(* IEC 61131-3 sources: POMIRTS_lab3/AS/Library_2/MTLoadSim/V1.01.0, 3 files *)

(* ---- MTLoadSim.typ ---- *)
(********************************************************************
 * COPYRIGHT -- Bernecker + Rainer
 ********************************************************************
 * Library: MTLoadSim
 * File: MTLoadSim.typ
 * Author: B + R
 ********************************************************************
 * Data types of library MTLoadSim
 ********************************************************************)

TYPE
	MTLoadSimConfigFrictionType : 	STRUCT
		Mode : MTLoadSimFricModeEnum;
		StaticFriction : REAL;
		DynamicFriction : REAL;
		ViscousFriction : REAL;
		StribeckVelocity : REAL;
		ApproximateVelocity : REAL;
		FrictionEpsilon : REAL;
		StribeckExponent : REAL;
	END_STRUCT;
	MTLoadSimConfigMassType : 	STRUCT
		Inertia : REAL;
		InitialStates : ARRAY[0..1]OF REAL;
	END_STRUCT;
	MTLoadSimConfigTwoMassType : 	STRUCT
		InertiaMass1 : REAL;
		InertiaMass2 : REAL;
		Stiff : REAL;
		Damp : REAL;
		Ratio : REAL;
		InitialStates : ARRAY[0..3]OF REAL;
	END_STRUCT;
	MTLoadSimMassConfigType : 	STRUCT
		Mass : MTLoadSimConfigMassType;
		Friction : MTLoadSimConfigFrictionType;
	END_STRUCT;
	MTLoadSimCouplConfigType : 	STRUCT
		Stiff : REAL;
		Damp : REAL;
		Ratio : REAL;
		Efficiency : REAL;
		BacklashWidth : REAL;
		InitialOutputBacklash : REAL;
	END_STRUCT;
	MTLoadSimStateValuesInternalType : 	STRUCT
		Position : LREAL;
		Velocity : LREAL;
		Acceleration : LREAL;
	END_STRUCT;
	MTLoadSimStateValuesType : 	STRUCT
		Position : LREAL;
		Velocity : REAL;
		Acceleration : REAL;
	END_STRUCT;
	MTLoadSimCouplInternalType : 	STRUCT
		TSample : REAL;
		Initialized : BOOL;
		InOperation : BOOL;
		Busy : BOOL;
		Error : BOOL;
		step : UINT;
		ErrorID : DINT;
		Position_old : LREAL;
		Configuration : MTLoadSimCouplConfigType;
		TorqueFeedback : LREAL;
		Torque : LREAL;
	END_STRUCT;
	MTLoadSimFricModeEnum :
		(
		mtLOADSIM_MODE_NO_FRICTION,
		mtLOADSIM_MODE_FRIC_KINETIC,
		mtLOADSIM_MODE_FRIC_KARNOPP,
		mtLOADSIM_MODE_FRIC_REGULATED
		);
	MTLoadSimFrictionInternalType : 	STRUCT
		TSample : REAL;
		Initialized : BOOL;
		InOperation : BOOL;
		Busy : BOOL;
		Error : BOOL;
		step : UINT;
		Reserve1 : UINT;
		ErrorID : DINT;
		Configuration : MTLoadSimConfigFrictionType;
		TorqueFriction : REAL;
	END_STRUCT;
	MTLoadSimTwoMassInternalType : 	STRUCT
		TSample : REAL;
		Initialized : BOOL;
		InOperation : BOOL;
		Busy : BOOL;
		Error : BOOL;
		Reserve1 : UINT;
		step : UINT;
		ErrorID : DINT;
		StateValuesMass1 : MTLoadSimStateValuesInternalType;
		Torque1 : LREAL;
		StateValuesMass2 : MTLoadSimStateValuesInternalType;
		Torque2 : LREAL;
		Configuration : MTLoadSimConfigTwoMassType;
		TorqueFriction : LREAL;
		SysVector : ARRAY[0..39]OF REAL;
		Reserve2 : UINT;
		StatusBusy : BOOL;
		StatusWorking : BOOL;
	END_STRUCT;
	MTLoadSimMassInternalType : 	STRUCT
		TSample : REAL;
		Initialized : BOOL;
		InOperation : BOOL;
		Busy : BOOL;
		Error : BOOL;
		step : UINT;
		Reserve1 : UINT;
		ErrorID : DINT;
		StateValues : MTLoadSimStateValuesInternalType;
		Configuration : MTLoadSimMassConfigType;
		TorqueFriction : REAL;
	END_STRUCT;
END_TYPE

(* ---- MTLoadSim.fun ---- *)
(********************************************************************
 * COPYRIGHT -- Bernecker + Rainer
 ********************************************************************
 * Library: MTLoadSim
 * File: MTLoadSim.fun
 * Author: B + R
 ********************************************************************
 * Functions and function blocks of library MTLoadSim
 ********************************************************************)

FUNCTION_BLOCK MTLoadSimCoupling
	VAR_INPUT
		Enable : BOOL;
		Configuration : MTLoadSimCouplConfigType;
		StateValues : MTLoadSimStateValuesType;
		StateValuesFeedback : MTLoadSimStateValuesType;
		ActivateSimulation : BOOL;
	END_VAR
	VAR_OUTPUT
		Initialized : BOOL;
		Busy : BOOL;
		Error : BOOL;
		ErrorID : DINT;
		Torque : REAL;
		TorqueFeedback : REAL;
		InOperation : BOOL;
	END_VAR
	VAR
		Internal : MTLoadSimCouplInternalType;
	END_VAR
END_FUNCTION_BLOCK

FUNCTION_BLOCK MTLoadSimMass
	VAR_INPUT
		Enable : BOOL;
		Configuration : MTLoadSimMassConfigType;
		Torque : REAL;
		TorqueFeedback : REAL;
		TorqueLoad : REAL;
		ActivateSimulation : BOOL;
	END_VAR
	VAR_OUTPUT
		Initialized : BOOL;
		Busy : BOOL;
		Error : BOOL;
		ErrorID : DINT;
		StateValues : MTLoadSimStateValuesType;
		StateValuesFeedback : MTLoadSimStateValuesType;
		InOperation : BOOL;
	END_VAR
	VAR
		Internal : MTLoadSimMassInternalType;
	END_VAR
END_FUNCTION_BLOCK

FUNCTION_BLOCK MTLoadSimFriction
	VAR_INPUT
		Enable : BOOL;
		Configuration : MTLoadSimConfigFrictionType;
		StateValues : MTLoadSimStateValuesType;
		StateValuesFeedback : MTLoadSimStateValuesType;
		TorqueDrive : REAL;
		ActivateSimulation : BOOL;
	END_VAR
	VAR_OUTPUT
		Initialized : BOOL;
		Busy : BOOL;
		Error : BOOL;
		ErrorID : DINT;
		TorqueFriction : REAL;
		InOperation : BOOL;
	END_VAR
	VAR
		Internal : MTLoadSimFrictionInternalType;
	END_VAR
END_FUNCTION_BLOCK

FUNCTION_BLOCK MTLoadSimTwoMass
	VAR_INPUT
		Enable : BOOL;
		Configuration : MTLoadSimConfigTwoMassType;
		Torque : REAL;
		TorqueFrictionMass1 : REAL;
		TorqueFrictionMass2 : REAL;
		TorqueLoad : REAL;
		ActivateSimulation : BOOL;
	END_VAR
	VAR_OUTPUT
		Initialized : BOOL;
		Busy : BOOL;
		Error : BOOL;
		ErrorID : DINT;
		StateValuesMass1 : MTLoadSimStateValuesType;
		StateValuesMass2 : MTLoadSimStateValuesType;
		StateValuesFeedback : MTLoadSimStateValuesType;
		TorqueMass1 : REAL;
		TorqueMass2 : REAL;
		InOperation : BOOL;
	END_VAR
	VAR
		Internal : MTLoadSimTwoMassInternalType;
	END_VAR
END_FUNCTION_BLOCK

(* ---- MTLoadSim.var ---- *)
(********************************************************************
 * COPYRIGHT -- Bernecker + Rainer
 ********************************************************************
 * Library: SimLoad
 * File: SimLoad.var
 * Author: B + R
 ********************************************************************
 * Constants of library SimLoad
 ********************************************************************)
VAR CONSTANT
	mtLOADSIM_ERR_INVALID_STIFFNESS : DINT := 1089667072;
	mtLOADSIM_ERR_INVALID_DAMPING : DINT := 1089667073;
	mtLOADSIM_ERR_INVALID_RATIO : DINT := 1089667074;
	mtLOADSIM_ERR_INVALID_EFFICIENCY : DINT := 1089667075;
	mtLOADSIM_ERR_INVALID_BACKLASH : DINT := 1089667076;
	mtLOADSIM_ERR_INVALID_TSAMPLE : DINT := 1089667077;
	mtLOADSIM_ERR_INVALID_ACTIVE : DINT := 1089667078;
	mtLOADSIM_ERR_INVALID_INERTIA : DINT := 1089667079;
	mtLOADSIM_ERR_INVALID_STAT_FRI : DINT := 1089667080;
	mtLOADSIM_ERR_INVALID_DYN_FRI : DINT := 1089667081;
	mtLOADSIM_ERR_INVALID_VISC_FRI : DINT := 1089667082;
	mtLOADSIM_ERR_INVALID_CHAR_VEL : DINT := 1089667083;
	mtLOADSIM_ERR_INVALID_FRIC_EPS : DINT := 1089667084;
	mtLOADSIM_ERR_INVALID_STRI_EXP : DINT := 1089667085;
	mtLOADSIM_ERR_INVALID_STRI_VEL : DINT := 1089667086;
	mtLOADSIM_ERR_INVALID_MODE : DINT := 1089667087;
	mtLOADSIM_ERR_INVALID_DATAPOINTS : DINT := 1089667088;
END_VAR
